FUNCTION_BLOCK FB_HMISimulationMotionRefGen
VAR_INPUT
END_VAR
VAR_OUTPUT
END_VAR
VAR
END_VAR

END_FUNCTION_BLOCK

(* stored: Version 1.1.0.1, ProductVersion 3.1.4024.10
   POU FB_HMISimulationMotionRefGen: Id {2af87d66-3ca9-458f-b958-0d830a205cdc}, SpecialFunc None *)
